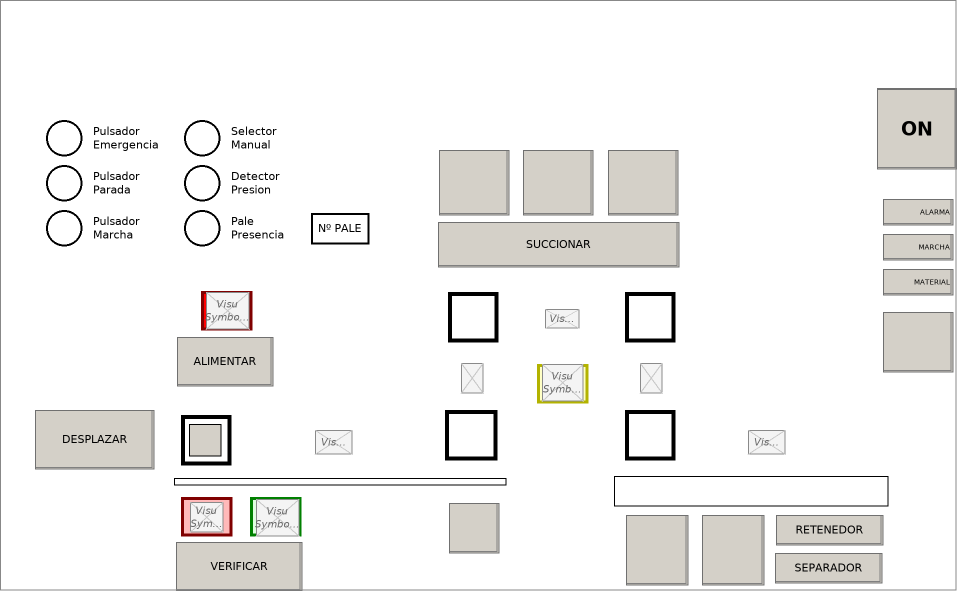
VISUALIZATION HMI_Proceso  // 957x591
    Rectangle (174,478 332x7)
    Rectangle (614,476 274x30)
    Button (176,542 126x49), "VERIFICAR"
        toggle MAIN.ESTACION.VerificadorBaja
    RoundedRectangle (250,497 51x39), colour toggle: MAIN.ESTACION.VerificadorAbajo
    RoundedRectangle (181,497 51x39), colour toggle: MAIN.ESTACION.VerificadorArriba
    Button (449,503 50x50), image: VisuSymbols.Symbols.Delete
        toggle MAIN.ESTACION.RechazadorAdelante
    Image (256,499 43x37), image: VisuSymbols.Symbols.OK
    Image (190,502 33x30), image: VisuSymbols.Symbols.Wrong
    Button (35,410 119x59), "DESPLAZAR"
        toggle MAIN.ESTACION.DesplazadorAdelante
    Rectangle (445,410 52x50)
        p4110469609: SEL(MAIN.ESTACION.DescargadorAtras AND MAIN.ESTACION.VerticalAbajo, 2, 0)
    Rectangle (181,415 50x50)
        p4110469609: SEL(MAIN.ESTACION.DesplazadorDetras, 2, 0)
    Rectangle (448,292 50x50)
        p4110469609: SEL((MAIN.ESTACION.DescargadorAtras AND MAIN.ESTACION.VerticalArriba), 2, 0)
    Rectangle (625,292 50x50)
        p4110469609: SEL(MAIN.ESTACION.DescargadorAdelante AND MAIN.ESTACION.VerticalArriba, 2, 0)
    Rectangle (625,410 50x50)
        p4110469609: SEL(MAIN.ESTACION.DescargadorAdelante AND MAIN.ESTACION.VerticalAbajo, 2, 0)
    Button (438,222 241x45), "SUCCIONAR"
        toggle MAIN.ESTACION.EyectorSucciona
    Button (439,150 70x65), image: VisuSymbols.Symbols.TriangleLeft
        tap MAIN.ESTACION.DescargadorAtras
    Button (523,150 70x65), image: VisuSymbols.Symbols.TriangleDown
        toggle MAIN.ESTACION.DescargadorBaja
    Button (608,150 70x65), image: VisuSymbols.Symbols.TriangleRight
        tap MAIN.ESTACION.DescargadorAdelante
    Image (545,309 34x19), image: VisuSymbols.Symbols.DoubleArrow3
    Image (640,363 22x30), image: VisuSymbols.Symbols.DoubleArrow4
    Image (461,363 22x30), image: VisuSymbols.Symbols.DoubleArrow4
    Image (315,430 37x24), image: VisuSymbols.Symbols.ArrowBoldRight
    Image (748,430 37x24), image: VisuSymbols.Symbols.ArrowBoldRight
    RoundedRectangle (201,291 51x39), colour toggle: MAIN.ESTACION.PresenciaBaseAlimentador
    RoundedRectangle (537,364 51x39), colour toggle: MAIN.ESTACION.VacioDescargador
    Image (542,364 41x37), image: VisuSymbols.Symbols.Caution
    Rectangle (190,425 30x30), invisible if: NotActivated(main.ESTACION.AlimentadorDelante)
    Image (216,296 24x30), invisible if: MAIN.ESTACION.PresenciaBaseAlimentador, image: Vacio.vacio
    Button (626,515 62x70), image: Vacio.onoff
        toggle MAIN.ESTACION.CintaMotorActiva
    Button (702,515 62x70), image: VisuSymbols.Symbols.ArrowCircle2RightUpDown
        tap MAIN.ESTACION.CintaMotorInvierte
    Button (776,515 107x30), "RETENEDOR"
        toggle MAIN.ESTACION.CintaRetenedorBaja
    Button (775,553 107x30), "SEPARADOR"
        toggle MAIN.ESTACION.CintaSeparadorSube
    Image (206,292 43x37), invisible if: NotActivated(main.ESTACION.PresenciaBaseAlimentador), image: VisuSymbols.Symbols.OK
    Button (877,88 80x80), "OFF", invisible if: MAIN.ESTACION.EstacionConectada
    Button (883,199 70x26), "ALARMA", image: VisuSymbols.Symbols.light
        toggle MAIN.ESTACION.LamparaAlarma
    Button (883,234 70x26), "MARCHA", image: VisuSymbols.Symbols.light
        toggle MAIN.ESTACION.LamparaMarcha
    Button (883,269 70x26), "MATERIAL", image: VisuSymbols.Symbols.light
        toggle MAIN.ESTACION.LamparaFaltaMaterial
    Button (883,312 70x60), image: VisuSymbols.Symbols.loudspeakerMedium
        toggle MAIN.ESTACION.AvisadorSonoro
    Rectangle (189,424 32x32), invisible if: not(MAIN.ESTACION.AlimentadorDetras)
    Button (177,337 96x49), "ALIMENTAR"
        toggle MAIN.ESTACION.AlimentadorAdelante
    Button (877,89 80x80), "ON", invisible if: NOT MAIN.ESTACION.EstacionConectada
        tap MAIN.ESTACION.DesconectaEstacion
    Ellipse (46,120 36x36), colour toggle: MAIN.ESTACION.PulsadorEmergencia
    Ellipse (46,165 36x36), colour toggle: MAIN.ESTACION.PulsadorParada
    Ellipse (46,210 36x36), colour toggle: MAIN.ESTACION.PulsadorMarcha
    Ellipse (184,120 36x36), colour toggle: MAIN.ESTACION.SelectorManual
    Ellipse (184,165 36x36), colour toggle: MAIN.ESTACION.DetectorPresion
    Label (90,123 83x30), "Pulsador Emergencia"
    Label (90,168 83x30), "Pulsador Parada"
    Label (90,213 83x30), "Pulsador Marcha"
    Label (228,123 83x30), "Selector Manual"
    Label (228,168 83x30), "Detector Presion"
    Ellipse (184,210 36x36), colour toggle: MAIN.ESTACION.PalePresencia
    Label (228,213 83x30), "Pale Presencia"
    Rectangle (311,213 58x31), "Nº PALE", text variable: MAIN.ESTACION.PaleCodigo
END_VISUALIZATION

(* stored: Version 1.1.0.1, ProductVersion 3.1.4024.12
   Visu HMI_Proceso: Id {6002bc90-4c57-4210-a85f-c15319348dec} *)
